PROGRAM Prozesskomponenten
VAR
	Bild_aufnehmen						:Skill_Bild_aufnehmen;
	Objekt_erkennen						:Skill_Objekt_erkennen;
	Greiferposition_ermitteln			:Skill_Greiferposition_ermitteln;
	
	Position_anfahren					:Skill_Position_anfahren;
	kontrolliert_bewegen				:Skill_Kontrolliert_bewegen;
	
	Backenposition_anfahren				:Skill_Backenposition_anfahren;
END_VAR

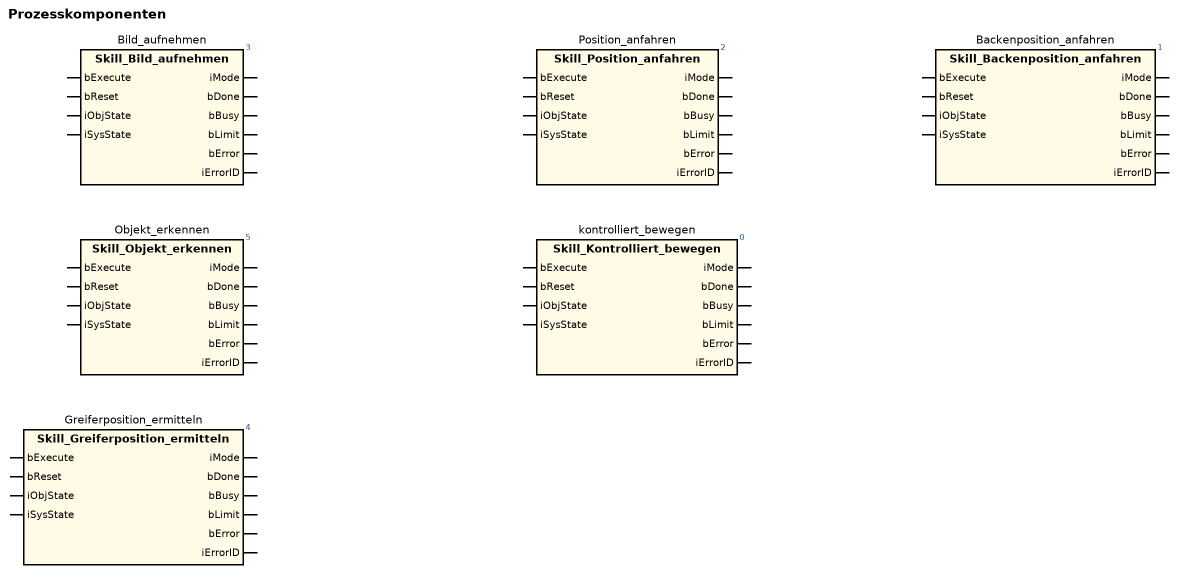
kontrolliert_bewegen(); // Skill_Kontrolliert_bewegen
Backenposition_anfahren(); // Skill_Backenposition_anfahren
Position_anfahren(); // Skill_Position_anfahren
Bild_aufnehmen(); // Skill_Bild_aufnehmen
Greiferposition_ermitteln(); // Skill_Greiferposition_ermitteln
Objekt_erkennen(); // Skill_Objekt_erkennen

END_PROGRAM

(* stored: Version 1.1.0.1
   POU Prozesskomponenten: Id {72d2be76-6370-4896-be86-f3be05fd5650}, SpecialFunc None *)
